Fanuc KAREL source: foo.kl

PROGRAM foo
%ALPHABETIZE
%COMMENT = ''
%NOBUSYLAMP
%NOLOCKGROUP
%NOPAUSE = COMMAND + TPENABLE + ERROR

%include lib_a\a.klt

%include klrdutil.kl


BEGIN
END foo
